FUNCTION_BLOCK FB_LogHandler_RetainableList EXTENDS FB_LogHandlerBase // Writes the last X-number of items to a retainable variable
VAR_OUTPUT PERSISTENT
	aLogItems : ARRAY[1..GVL_Utilities.RETAINABLE_LOG_HISTORY_SIZE] OF UDT_LogItem;
	nIndex : UINT; // Index in the array of the last added log item
END_VAR

METHOD INTERNAL FINAL AddToLog
VAR_INPUT
	stLogItem : UDT_LogItem;
END_VAR
VAR
	i : UINT; // Iterator
END_VAR
nIndex := (nIndex MOD GVL_Utilities.RETAINABLE_LOG_HISTORY_SIZE) + 1;
aLogItems[nIndex] := stLogItem;
END_METHOD

END_FUNCTION_BLOCK

(* stored: Version 1.1.0.1, ProductVersion 3.1.4024.11
   POU FB_LogHandler_RetainableList: Id {4966cdb4-950f-0659-2a45-e07380f91fca}, SpecialFunc None
   Method AddToLog: Id {10aa411e-05f8-09bd-04b5-bb2a775a1d6a} *)
